(* IEC 61131-3 sources: rust-plc/playground/oop_project/classes, 3 files *)

(* ---- alarm.st ---- *)
(*
 * Alarm class — monitors a value and triggers on threshold.
 * Uses pointer-based output pattern to write status to caller.
 *)

CLASS Alarm IMPLEMENTS IResettable
VAR
    _active    : BOOL := FALSE;
    _limit     : INT := 100;
    _hyst      : INT := 5;
    _tripCount : INT := 0;
END_VAR

    PUBLIC METHOD Configure
    VAR_INPUT limit : INT; hyst : INT; END_VAR
        _limit := limit;
        _hyst := hyst;
    END_METHOD

    PUBLIC METHOD Evaluate
    VAR_INPUT value : INT; END_VAR
    VAR wasActive : BOOL; END_VAR
        wasActive := _active;
        IF value > _limit THEN
            _active := TRUE;
        ELSIF value < (_limit - _hyst) THEN
            _active := FALSE;
        END_IF;
        IF _active AND NOT wasActive THEN
            _tripCount := _tripCount + 1;
        END_IF;
    END_METHOD

    PUBLIC METHOD IsActive : INT
        IF _active THEN IsActive := 1; ELSE IsActive := 0; END_IF;
    END_METHOD

    PUBLIC METHOD GetTripCount : INT
        GetTripCount := _tripCount;
    END_METHOD

    PUBLIC METHOD WriteStatus
    VAR_INPUT pActive : REF_TO INT; pTrips : REF_TO INT; END_VAR
        IF pActive <> NULL THEN
            IF _active THEN pActive^ := 1; ELSE pActive^ := 0; END_IF;
        END_IF;
        IF pTrips <> NULL THEN pTrips^ := _tripCount; END_IF;
    END_METHOD

    PUBLIC METHOD Reset
        _active := FALSE;
        _tripCount := 0;
    END_METHOD
END_CLASS

(* ---- controller.st ---- *)
(*
 * Controller classes — base and derived.
 * Demonstrates cross-file inheritance: BaseController → TempController.
 * Uses IControllable interface from interfaces/.
 * Uses Clamp from utils/.
 *)

CLASS BaseController IMPLEMENTS IControllable
VAR
    _enabled : BOOL := FALSE;
    _output  : INT := 0;
END_VAR

    PUBLIC METHOD Enable
        _enabled := TRUE;
    END_METHOD

    PUBLIC METHOD Disable
        _enabled := FALSE;
        _output := 0;
    END_METHOD

    PUBLIC METHOD IsEnabled : INT
        IF _enabled THEN IsEnabled := 1; ELSE IsEnabled := 0; END_IF;
    END_METHOD

    PUBLIC METHOD GetOutput : INT
        GetOutput := _output;
    END_METHOD
END_CLASS

CLASS TempController EXTENDS BaseController IMPLEMENTS IResettable
VAR
    _setpoint   : INT := 50;
    _gain       : INT := 20;
    _outMin     : INT := 0;
    _outMax     : INT := 100;
END_VAR

    PUBLIC METHOD Configure
    VAR_INPUT
        sp   : INT;
        gain : INT;
        oMin : INT;
        oMax : INT;
    END_VAR
        _setpoint := sp;
        _gain := gain;
        _outMin := oMin;
        _outMax := oMax;
    END_METHOD

    PUBLIC METHOD Compute
    VAR_INPUT pv : INT; END_VAR
    VAR error : INT; raw : INT; END_VAR
        IF _enabled THEN
            error := _setpoint - pv;
            raw := (error * _gain) / 10;
            _output := Clamp(val := raw, lo := _outMin, hi := _outMax);
        ELSE
            _output := 0;
        END_IF;
    END_METHOD

    PUBLIC METHOD GetSetpoint : INT
        GetSetpoint := _setpoint;
    END_METHOD

    PUBLIC METHOD Reset
        _output := 0;
        _enabled := FALSE;
    END_METHOD
END_CLASS

(* ---- sensor.st ---- *)
(*
 * Sensor class — reads and filters analog input.
 * Implements IResettable.
 * Uses Clamp from utils/math_utils.st.
 *)

CLASS Sensor IMPLEMENTS IResettable
VAR
    _raw      : INT := 0;
    _filtered : INT := 0;
    _count    : INT := 0;
    _min      : INT := 32767;
    _max      : INT := 0;
END_VAR

    PUBLIC METHOD Update
    VAR_INPUT rawValue : INT; END_VAR
    VAR clamped : INT; END_VAR
        clamped := Clamp(val := rawValue, lo := 0, hi := 1000);
        _raw := clamped;
        // Simple EMA filter: 25% new + 75% old
        IF _count = 0 THEN
            _filtered := clamped;
        ELSE
            _filtered := (25 * clamped + 75 * _filtered) / 100;
        END_IF;
        _count := _count + 1;
        IF clamped < _min THEN _min := clamped; END_IF;
        IF clamped > _max THEN _max := clamped; END_IF;
    END_METHOD

    PUBLIC METHOD GetFiltered : INT
        GetFiltered := _filtered;
    END_METHOD

    PUBLIC METHOD GetRaw : INT
        GetRaw := _raw;
    END_METHOD

    PUBLIC METHOD GetMin : INT
        GetMin := _min;
    END_METHOD

    PUBLIC METHOD GetMax : INT
        GetMax := _max;
    END_METHOD

    PUBLIC METHOD GetSampleCount : INT
        GetSampleCount := _count;
    END_METHOD

    PUBLIC METHOD Reset
        _raw := 0;
        _filtered := 0;
        _count := 0;
        _min := 32767;
        _max := 0;
    END_METHOD
END_CLASS
